% RSLogix 500 project practice.RSS, saved by version 8.30.00.16 %
PROJECT "UNTITLED"    % processor: MicroLogix 1000 %

PROGRAM FILES
  LAD 2 "MAIN_PROG"  5 rungs
  LAD 3 "USER_FAULT"  1 rungs
  LAD 4 "HSC_INT"  1 rungs
  LAD 5 "STI_INT"  1 rungs
  LAD 6, 7, 8, 9, 10, 11, 12, 13, 14, 15, 16: only END

DATA FILES
  O0 OUTPUT  1 elements
  I1 INPUT  2 elements
  S2 STATUS  33 elements
  B3 BINARY  32 elements
  T4 TIMER  40 elements
  C5 COUNTER  32 elements
  R6 CONTROL  16 elements
  N7 INTEGER  105 elements

LADDER 2 "MAIN_PROG"
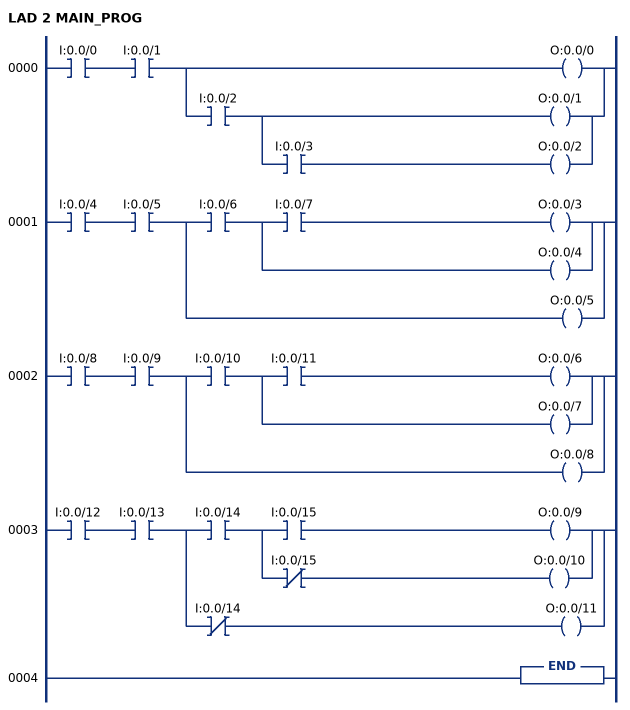
% Rung: 0 %
SOR XIC I:0.0/0 XIC I:0.0/1 BST OTE O:0.0/0 NXB XIC I:0.0/2 BST OTE O:0.0/1 NXB XIC I:0.0/3 OTE O:0.0/2 BND BND EOR
% Rung: 1 %
SOR XIC I:0.0/4 XIC I:0.0/5 BST XIC I:0.0/6 BST XIC I:0.0/7 OTE O:0.0/3 NXB OTE O:0.0/4 BND NXB OTE O:0.0/5 BND EOR
% Rung: 2 %
SOR XIC I:0.0/8 XIC I:0.0/9 BST XIC I:0.0/10 BST XIC I:0.0/11 OTE O:0.0/6 NXB OTE O:0.0/7 BND NXB OTE O:0.0/8 BND EOR
% Rung: 3 %
SOR XIC I:0.0/12 XIC I:0.0/13 BST XIC I:0.0/14 BST XIC I:0.0/15 OTE O:0.0/9 NXB XIO I:0.0/15 OTE O:0.0/10 BND NXB XIO I:0.0/14 OTE O:0.0/11 BND EOR
% Rung: 4 %
SOR END EOR
